DATA_BLOCK "BalanceTank_DB"
{ S7_Optimized_Access := 'TRUE' }
"FB_BalanceTank"


BEGIN

END_DATA_BLOCK
